	20:		(* Move to idle *)
		uiSignalOutControl := Move_to_idle;
		IF uiSignalInAck = Move_to_idle THEN
			uiSignalOutControl := 0;
			NewState := 25;
		END_IF

	25:
		IF uiSignalInAck = 0 THEN
			NewState := 30;
		END_IF

	30:		(* Set CmdByte to 2, to tell PC to start calibration of Cam 1 *)
		bCalibCamOneStart := TRUE;

		IF stDataFromVision.CmdInProcess =  stDataToVision.CmdByte AND stDataToVision.CmdByte <> 0 THEN							(* When PC recieve command, it sends acknowledge *)
			bCalibCamOneStart := FALSE;
			NewState := 35;
		END_IF
		
	35:
		FB_CLOSE_CUT.Execute := TRUE;
		IF FB_CLOSE_CUT.Done THEN
			FB_CLOSE_CUT.Execute := FALSE;
			NewState := 37;
		END_IF
		
	37:
		IF sNewCalib = 'calib-mounted' THEN
			NewState := 40;
		END_IF
		

	40:		(* Call CALIB_CAM1 on robot Cut. Robot Cut move to a pos to take a picture *)
		uiSignalOutControl := CalibCamOne;
		IF uiSignalInAck = CalibCamOne THEN
			uiSignalOutControl := 0;
			NewState := 45;
		END_IF

	45:
		IF uiSignalInAck = 0 THEN
			NewState := 50;
		END_IF

	50:		(* Before the picture is taken, call get cut coord *)
		getCutCoords := TRUE;										(* Get coord from robot Cut *)
		IF uiSignalInAck = getCurrentCutCoords THEN
			uiSignalOutControl := 0;
			NewState := 55;
		END_IF

	55:
		IF uiSignalInAck = 0 THEN
			bWait := TRUE;
			IF Wait.Q THEN
				bWait := FALSE;
				NewState := 60;
			END_IF
		END_IF

	60:		(* CmdByte 3 means that we want to take a picture *)
		bNewPosCalibCamOne := TRUE;
		IF stDataFromVision.CmdInProcess =  stDataToVision.CmdByte AND stDataToVision.CmdByte <> 0 THEN
			bNewPosCalibCamOne := FALSE;
			NewState := 70;
		END_IF

	70:		(* If there has not been taken enough pictures go to state 40 in order to take more picture. Else send CmdByte 4 to tell PC to stop calib *)
		uiCalibImgCount := uiCalibImgCount + 1;
		IF uiCalibImgCount < 8 THEN
			NewState := 40;
		ELSE
			uiCalibImgCount := 0;
			bEndCalibCamOne := TRUE;
			NewState := 80;
		END_IF

	80:		(* Reset CmdByte and go to init state *)
		uiSignalOutControl := Move_to_idle;
		IF uiSignalInAck = Move_to_idle THEN
			uiSignalOutControl := 0;
			NewState := 82;
		END_IF
	
	82:		
		IF sNewCalib = 'calib-unmounted' THEN
			uiSignalOutTool.06 := FALSE;
			NewState := 84;
		END_IF	
		
	84:
		uiSignalOutControl := Move_to_idle;
		IF uiSignalInAck = Move_to_idle THEN
			uiSignalOutControl := 0;
			NewState := 90;
		END_IF

	85:
		IF uiSignalInAck = 0 THEN
			NewState := 90;
		END_IF

	90:
		IF stDataFromVision.CmdInProcess = stDataToVision.CmdByte AND stDataToVision.CmdByte <>0 THEN
			bEndCalibCamOne := FALSE;
			GbCloseCut := FALSE;
			uiStatus := 0;
			NewState := 0;
		END_IF

	1000:		(* RESET *)
		uiSignalOutTool.06 := FALSE;
		startCalibCam1 			:= FALSE;
		uiSignalOutControl 		:= 0;
		bCalibCamOneStart 		:= FALSE;
		getCutCoords				:= FALSE;
		bNewPosCalibCamOne 	:= FALSE;
		uiCalibImgCount			:= 0;
		bEndCalibCamOne		:= FALSE;

		NewState := 0;

	2000:
		bStopped := TRUE;


END_CASE

IF bStart AND NOT bStop AND NOT bAlarmState AND uiprogNo = 1 AND State <> 2000 THEN
	startCalibCam1 := TRUE;
	(*bStart := FALSE;*)
	uiStatus := 1;
END_IF

IF State <> 2000 THEN
	bStopped := FALSE;
END_IF
Wait		(IN:=  bWait		, PT:=t#1000ms, Q=>, ET=>); 		(*Timer*)
Wait2	(IN:=  bWait2		, PT:=t#2000ms, Q=>, ET=>); 	(*Timer*)
Wait3	(IN:=  bWait3		, PT:=t#2000ms, Q=>, ET=>); 	(*Timer*)

END_PROGRAM

// ---- POUs/CONTROLs/CalibCam2.TcPOU
PROGRAM CalibCam2
VAR_INPUT
	State: INT :=0;
	NewState: INT := 0;
END_VAR

VAR

	Wait: TON;
	Wait2: TON;
	bWait: BOOL;
	bWait2: BOOL;
	next: BOOL;
	Wait3: TON;
	bWait3: BOOL;
	flag: BOOL;
	bStopped: BOOL;
END_VAR

IF sNewCalib = 'he-pick-start' THEN
	startCalibCam2 := TRUE;
ELSE
	startCalibCam2 := FALSE;
END_IF

CASE State OF

	0:		(* Init State - Wait for Calibration of camera 2 *)
		uiSignalOut3.01 := FALSE;
		IF (uiprogNo = 2 OR allZero) AND startCalibCam2 AND State <> 2000  AND NOT bAlarmState THEN
			bWait2 := FALSE;
			uiCalibImgCount := 0;
			uiSignalOut3.01 := TRUE;								(* Tells robot Cut to move to Calib cam 2 pos *)
			startCalibCam2 := FALSE;
			uiSignalOutTool.06 := TRUE;
			flag := FALSE;
			NewState := 10;
		END_IF

	10:		(* Set velocity *)
		uiSignalOutSpeedControl := UINT_TO_BYTE(uiSpeedSetting);
		uiSignalOutControl := Set_Velocity;
		IF uiSignalInAck = Set_Velocity THEN
			uiSignalOutControl := 0;
			NewState := 15;
		END_IF

	15:
		IF uiSignalInAck = 0 THEN
			NewState := 20;
		END_IF

	20:		(* Move to idle *)
		uiSignalOutControl := Move_to_idle;
		IF uiSignalInAck = Move_to_idle THEN
			uiSignalOutControl := 0;
			NewState := 25;
		END_IF

	25:
		IF uiSignalInAck = 0 THEN
			NewState := 27;
		END_IF
		
	27: 		
		FB_CLOSE_CUT.Execute := TRUE;
		IF FB_CLOSE_CUT.Done THEN
			FB_CLOSE_CUT.Execute := FALSE;
			NewState := 29;
		END_IF
	
	29:
		IF sNewCalib = 'calib-mounted' THEN
			NewState := 30;
		END_IF

	30:		(* Move Robot cut to pos for calib *)
		uiSignalOutControl := CalibCamOne;
		IF uiSignalInAck = CalibCamOne THEN
			uiSignalOutControl := 0;
			NewState := 35;
		END_IF

	35:
		IF uiSignalInAck = 0 THEN
			NewState := 40;
		END_IF

	40:		(* Get robot cut pos and orientation *)
		getCutCoords := TRUE;
		IF bPosSentToPcCom AND FB_GET_CUT_COORD.Execute = FALSE THEN
			IF stDataToVision.CoordXR1G <> 0 THEN
				bPosSentToPcCom := FALSE;
				gResetPcCom := TRUE;
				NewState := 45;
			END_IF
		END_IF

	45:
		IF uiSignalInAck = 0 THEN
			GviX	:= stDataToVision.CoordXR1G / 10;
			GviY	:= stDataToVision.CoordYR1G / 10;
			GviZ	:= stDataToVision.CoordZR1G / 10;
			GviA	:= - currentRobotA;
			GviE	:= - currentRobotE;
			GviR	 := 60;
			gResetPcCom := TRUE;

			NewState := 50;
		END_IF

	50:		(* Sends coordinates of calibration board to robot pick *)

		bCalibCamTwoStart := TRUE;
		(* GsendCoord			-->	Starter SendCoordinates sekvensen							-	Sender koordinater til robotterne 		*)
		(* uiSignalOutShared.06	-->	Bekræftelse på at koordinaterne er sendt til udgangene i box 10	-	Acknowledge fra SendCoordinates	*)
		GsendCoord := TRUE;
		IF uiSignalOutShared.06 THEN
			(* Send_pos	-->	Kommando der fortæller robot cut at nogle nye positioner er sendt *)
			uiSignalOutControl := Send_pos;
		END_IF
		IF uiSignalInAck = Send_pos THEN
			uiSignalOutControl := 0;
			NewState := 55;
		END_IF

	55:
		IF uiSignalInAck = 0 THEN
			IF stDataFromVision.CmdInProcess =  stDataToVision.CmdByte AND stDataToVision.CmdByte <> 0 THEN
				bCalibCamTwoStart := FALSE;
				gResetPcCom := TRUE;
				NewState := 60;
			END_IF
		END_IF

	60:		(* Call CALIB_CAM2 on robot Pick. This means that robot Pick move to a pos so that the camera can take a picture *)
		uiSignalOutControl := CalibCamTwo;

		IF uiSignalInAck = CalibCamTwo THEN
			uiSignalOutControl := 0;
			NewState := 65;
		END_IF

	65:
		IF uiSignalInAck = 0 THEN
			NewState := 70;
		END_IF

	70:		(* Before the picture is taken, call get pick coord *)
		getPickCoords := TRUE;
		IF uiSignalInAck = getCurrentPickCoords THEN
			uiSignalOutControl := 0;
			NewState := 75;
		END_IF

	75:
		IF uiSignalInAck = 0 THEN
			bWait2 := TRUE;
			IF Wait2.Q THEN
				bWait2 := FALSE;
				NewState := 80;
			END_IF
		END_IF

	80:		(* CmdByte 6 means that we want to take a picture *)
		IF next5 THEN
			bNewPosCalibCamTwo := TRUE;
			IF stDataFromVision.CmdInProcess =  stDataToVision.CmdByte AND stDataToVision.CmdByte <> 0  THEN
				next5 := FALSE;
				bNewPosCalibCamTwo := FALSE;
				NewState := 85;
			END_IF
		END_IF

	85:		(* If there has not been taken enough pictures go to state 40 in order to take more picture. Else send CmdByte 7 to tell PC to stop calib *)
		uiCalibImgCount := uiCalibImgCount + 1;
		IF uiCalibImgCount < 11 THEN
			gResetPcCom := TRUE;
			NewState := 60;	(* 40 Before *)
		ELSE
			uiCalibImgCount := 0;
			bEndCalibCamTwo := TRUE;
			NewState := 86;
		END_IF
		
	86:
		FB_PICK_TO_IDLE.Execute := TRUE;
		uiSignalOutControl := FB_PICK_TO_IDLE.OutQ;
		IF FB_PICK_TO_IDLE.Done THEN
			FB_PICK_TO_IDLE.Execute := FALSE;
			NewState := 87;
		END_IF
		
	87:
		FB_CUT_TO_IDLE.Execute := TRUE;
		uiSignalOutControl := FB_CUT_TO_IDLE.OutQ;
		IF FB_CUT_TO_IDLE.Done THEN
			IF stDataFromVision.CmdInProcess = stDataToVision.CmdByte  AND stDataToVision.CmdByte <> 0 THEN
				FB_CUT_TO_IDLE.Execute := FALSE;
				bEndCalibCamTwo := FALSE;
				uiStatus := 0;
				uiSignalOutTool.06 := FALSE;
				NewState := 88;
			END_IF
		END_IF
		
	88:
		IF sNewCalib = 'calib-unmounted' THEN
			NewState := 90;
		END_IF	
		

	90:		(* Reset CmdByte and go to init state *)
		//bBackToZero := TRUE;
		uiSignalOutControl := Move_to_idle;
		IF uiSignalInAck = Move_to_idle AND NOT bAck THEN
			uiSignalOutControl := 0;
			IF stDataFromVision.CmdInProcess = stDataToVision.CmdByte  AND stDataToVision.CmdByte <> 0 THEN
				bEndCalibCamTwo := FALSE;
				uiStatus := 0;
				NewState := 95;
			END_IF
		END_IF
		
	95:
		IF uiSignalInAck = 0 THEN
			PcCom.state := 0;
			NewState := 0;
		END_IF

	1000: 		(* RESET *)
		uiSignalOutTool.06 		:= FALSE;
		uiSignalOut3.01 			:= FALSE;
		startCalibCam2 			:= FALSE;
		flag 						:= FALSE;
		uiSignalOutControl 		:= 0;
		getCutCoords 			:= FALSE;
		getPickCoords 			:= FALSE;
		bCalibCamTwoStart 		:= FALSE;
		GcoordSent 				:= FALSE;
		bNewPosCalibCamTwo 	:= FALSE;
		next5 					:= FALSE;
		uiCalibImgCount 			:= 0;
		bEndCalibCamTwo 		:= FALSE;
		bWait2 					:= FALSE;

		NewState := 0;

	2000:
		bStopped := TRUE;


END_CASE

IF bStart AND NOT bStop AND NOT bAlarmState AND uiprogNo = 2 AND State <> 2000 THEN
	startCalibCam2 := TRUE;
	bStart := FALSE;
	uiStatus := 1;
END_IF

IF State <> 2000 THEN
	bStopped := FALSE;
END_IF

Wait		(IN:=  bWait		, PT:=t#200ms, Q=>, ET=>); 		(*Timer*)
Wait2	(IN:=  bWait2		, PT:=t#2000ms, Q=>, ET=>); 	(*Timer*)
Wait3	(IN:=  bWait3		, PT:=t#2000ms, Q=>, ET=>); 	(*Timer*)

END_PROGRAM

// ---- POUs/BackToZero.TcPOU
PROGRAM BackToZero
VAR_INPUT
	State: 		INT := 0;
	NewState:	INT := 0;
END_VAR
VAR
	uiPickCoordX: UINT;
	uiPickCoordY: UINT;
	uiPickCoordZ: UINT;
	
	flag: bool := false;

	StartBackToZero: BOOL;
	bReset: BOOL;
	CANCEL_MOVE: BOOL;
	uiCutCoordX: UINT;
	uiCutCoordY: UINT;
	uiCutCoordZ: UINT;

	timer : TON;
	CoordZR2G: INT;
	PICKMOVED: BOOL;
	CUTMOVED: BOOL;
	whatState: INT;
END_VAR

(* Start connection to Robot Cut if physical botton or HMI button is pressed *)
IF bBackToZero THEN
	StartBackToZero := TRUE;
ELSE
	StartBackToZero := FALSE;
END_IF

CASE State OF

	0:
		IF StartBackToZero THEN
			NewState  	:= 10;
		END_IF

	10:		(* RESET ALL SEQUENCES *)
		IF NOT bReset THEN
			whatState :=  Control.State;
			bReset := TRUE;
			BlockTest.				NewState := 1000;
			Control.					NewState := 1000;
			ControlAuto.				NewState := 1000;
			ControlMoveToCalibPos.	NewState := 1000;
			CalibCam1.				NewState := 1000;
			CalibCam2.				NewState := 1000;
			ControlGrabAuto.			NewState := 1000;

			FB_GET_STEM.			NewState := 1000;
			FB_GRAB_STEM.			NewState := 1000;
			FB_MOVE_ON_STEM.		NewState := 1000;
			FB_FIND_JOINT.			NewState := 1000;
			FB_GRAB_JOINT.			NewState := 1000;
			FB_DELEAF_PLACE.		NewState := 1000;

			getPickCoords 	:= FALSE;
			getCutCoords 	:= FALSE;
		END_IF

		IF Control.NewState = 0 AND ControlAuto.NewState = 0 AND ControlMoveToCalibPos.NewState = 0 AND
			CalibCam1.NewState = 0 AND CalibCam2.NewState = 0 AND ControlGrabAuto.NewState = 0 THEN
			timer.IN := TRUE;
			IF timer.Q THEN
				timer.IN := FALSE;
				bReset := FALSE;
				getPickCoords := FALSE;
				getCutCoords := FALSE;
				NewState := 20;
			END_IF
		END_IF

	20:		(* SEND SIGNAL TO ROBOTS TO STOP MOTION *)
		CANCEL_MOVE := TRUE;
		IF uiSignalInAck = 0 THEN
			timer.IN := TRUE;
			IF timer.Q THEN
				timer.IN := FALSE;
				CANCEL_MOVE := FALSE;
				NewState := 25;
			END_IF
		END_IF
		
	25:		(* Set calibration velocity *)
		uiSignalOutSpeedControl := UINT_TO_BYTE(uiSpeedSetting);
		uiSignalOutControl := Set_Velocity;

		IF uiSignalInAck = Set_Velocity THEN
			uiSignalOutControl := 0;
			NewState := 30;
		END_IF


	30:		(* FIGURE OUT WHICH ROBOT IS SITURATED THE LOWEST *)
		(* Get Cut coord *)
		getCutCoords := TRUE;
		IF bPosSentToPcCom AND FB_GET_CUT_COORD.Execute = FALSE THEN
			bPosSentToPcCom := FALSE;
			gResetPcCom := TRUE;
			NewState := 35;
		END_IF

	35:
		IF uiSignalInAck = 0 THEN
			uiCutCoordX	:= stDataToVision.CoordXR1G / 10;
			uiCutCoordY	:= stDataToVision.CoordYR1G / 10;
			uiCutCoordZ	:= stDataToVision.CoordZR1G / 10;
			timer.IN := TRUE;
			IF timer.Q THEN
				timer.IN := FALSE;
				gResetPcCom := TRUE;
				NewState := 40;
			END_IF
		END_IF


	40:
		(* Get Cut coord *)
		getPickCoords := TRUE;
		IF bPosSentToPcCom AND FB_GET_PICK_COORD.Execute = FALSE THEN
			bPosSentToPcCom := FALSE;
			gResetPcCom := TRUE;
			NewState := 45;
		END_IF

	45:
		IF uiSignalInAck = 0 THEN
			uiPickCoordX	:= stDataToVision.CoordXR2G / 10;
			uiPickCoordY	:= stDataToVision.CoordYR2G / 10;
			uiPickCoordZ	:= stDataToVision.CoordZR2G / 10;
			timer.IN := TRUE;
			IF timer.Q THEN
				timer.IN := FALSE;
				gResetPcCom := TRUE;
				NewState := 50;
			END_IF
		END_IF
		
	50:		(* MOVE THE FIRST ROBOT AWAY *)
		IF whatState >= 400 AND whatState <=500 THEN
			FB_PICK_TO_ZERO.Execute := TRUE;
			uiSignalOutControl := FB_PICK_TO_ZERO.OutQ;
			IF FB_PICK_TO_ZERO.Done THEN
				PICKMOVED := TRUE;
				FB_PICK_TO_ZERO.Execute := FALSE;
				NewState := 60;
			END_IF
		ELSE
			FB_CUT_TO_ZERO.Execute := TRUE;
			uiSignalOutControl := FB_CUT_TO_ZERO.OutQ;
			IF FB_CUT_TO_ZERO.Done THEN
				CUTMOVED := TRUE;
				FB_CUT_TO_ZERO.Execute := FALSE;
				NewState := 60;
			END_IF
		END_IF

	60:		(* MOVE THE LAST ROBOT *)
		IF PICKMOVED THEN
			FB_CUT_TO_ZERO.Execute := TRUE;
			uiSignalOutControl := FB_CUT_TO_ZERO.OutQ;
			IF FB_CUT_TO_ZERO.Done THEN
				FB_CUT_TO_ZERO.Execute := FALSE;
				NewState := 70;
			END_IF
		ELSE
			FB_PICK_TO_ZERO.Execute := TRUE;
			uiSignalOutControl := FB_PICK_TO_ZERO.OutQ;
			IF FB_PICK_TO_ZERO.Done THEN
				FB_PICK_TO_ZERO.Execute := FALSE;
				NewState := 70;
			END_IF
		END_IF

	(*50:		(* MOVE THE LOWEST ROBOT AWAY *)
		IF uiCutCoordZ < (uiPickCoordZ - 20) THEN
			FB_CUT_TO_ZERO.Execute := TRUE;
			uiSignalOutControl := FB_CUT_TO_ZERO.OutQ;
			IF FB_CUT_TO_ZERO.Done THEN
				FB_CUT_TO_ZERO.Execute := FALSE;
				NewState := 60;
			END_IF
		ELSE
			FB_PICK_TO_ZERO.Execute := TRUE;
			uiSignalOutControl := FB_PICK_TO_ZERO.OutQ;
			IF FB_PICK_TO_ZERO.Done THEN
				FB_PICK_TO_ZERO.Execute := FALSE;
				NewState := 60;
			END_IF
		END_IF

	60:		(* MOVE THE LAST ROBOT *)
		IF uiCutCoordZ > (uiPickCoordZ - 20) THEN
			FB_CUT_TO_ZERO.Execute := TRUE;
			uiSignalOutControl := FB_CUT_TO_ZERO.OutQ;
			IF FB_CUT_TO_ZERO.Done THEN
				FB_CUT_TO_ZERO.Execute := FALSE;
				NewState := 70;
			END_IF
		ELSE
			FB_PICK_TO_ZERO.Execute := TRUE;
			uiSignalOutControl := FB_PICK_TO_ZERO.OutQ;
			IF FB_PICK_TO_ZERO.Done THEN
				FB_PICK_TO_ZERO.Execute := FALSE;
				NewState := 70;
			END_IF
		END_IF*)

	70:		(* MOVE BACK TO IDLE *)
		FB_MOVE_TO_IDLE.Execute := TRUE;
		uiSignalOutControl := FB_MOVE_TO_IDLE.OutQ;
		IF FB_MOVE_TO_IDLE.Done THEN
			FB_MOVE_TO_IDLE.Execute := FALSE;
			NewState := 80;
		END_IF


	80:		(* RESET THE TOOLS *)
		IF flag = FALSE THEN
			Tools.NewState := 1000;
			flag := TRUE;
		END_IF
		
		IF uiToolState = 0 THEN
			flag := false;
			NewState := 90;
		END_IF


	90:		(* RESET VALUES AND CHANGE STATE TO 0 *)
		bBackToZero := FALSE;
		CANCEL_MOVE := FALSE;
		PICKMOVED := FALSE;
		CUTMOVED := FALSE;
		whatState := 0;

		uiCutCoordX	:= 0;
		uiCutCoordY	:= 0;
		uiCutCoordZ 	:= 0;
		uiPickCoordX	:= 0;
		uiPickCoordY := 0;
		uiPickCoordZ := 0;
		gStopped := TRUE;
		NewState := 0;


END_CASE

uiSignalOut2.03 := CANCEL_MOVE;
 timer( PT:=t#500ms, Q=>, ET=>);

END_PROGRAM

// ---- POUs/CONTROLs/BlockTest.TcPOU
PROGRAM BlockTest
VAR_INPUT
	State: INT := 0;
	NewState: INT := 0;

	InternalState: INT := 0;
	InternalNewState: INT := 0;
END_VAR

VAR
	(* FUNCTION BLOCKS *)
	(*FB_PLACE: 		PlaceCoordinates;
	FB_GET_STEM:	GetStem;*)

	(* REALS *)

	(* INTEGERS *)


	ImageRetryHeight:	INT;

	iMoved: 			INT;					(* Hvor mange gange har cut bevæget sig efter iBunchPosZ er nået *)
	iCnfgChange:		INT := 0;
	uiDeleaf: 		UINT;

	(* BOOLS *)
	bStopped: BOOL;
	bRobotFail: BOOL;

	bRetry: INT;
	bStemGrabbed: BOOL;

END_VAR

CASE State OF

	0:		(* init	-	Every important variables will be resat before the start of the sequence *)
		IF bStart AND uiprogNo = 7 AND State <> 2000  AND NOT bAlarmState THEN
			uiStatus := 1;

			(* Init variables *)
			bRetry := 0;
			uiCalibImgCount	:= 0;
			iMoved := 0;
			iImageZone := 0;
			gJointFound := 0;
			gResetPcCom 	:= TRUE;
			iCnfgChange := 0;
			uiDeleaf := 0;
			bPosSentToPcCom := FALSE;

			(* Before starting - Home *)
			GbHomeGripStem := TRUE;
			IF bHomeDone THEN
				bStart := FALSE;
				bHomeDone := FALSE;
				NewState := 10;
			END_IF
		END_IF

	10:		(* Set velocity *)
		FB_SET_VELOCITY.Execute := TRUE;
		uiSignalOutSpeedControl := UINT_TO_BYTE(uiSpeedSetting);
		uiSignalOutControl := FB_SET_VELOCITY.OutQ;
		IF FB_SET_VELOCITY.Done THEN
			FB_SET_VELOCITY.Execute := FALSE;
			NewState := 20;
		END_IF

	20:		(* Idle *)
		FB_MOVE_TO_IDLE.Execute := TRUE;
		uiSignalOutControl := FB_MOVE_TO_IDLE.OutQ;
		IF FB_MOVE_TO_IDLE.Done THEN
			FB_MOVE_TO_IDLE.Execute := FALSE;
			NewState := 30;
		END_IF




		(* ------------------------------------------------------------------- Get Stem  ------------------------------------------------------------------- *)
	30:				(*  Load cutter *)
		FB_LOAD_CUT.Execute := TRUE;
		IF FB_LOAD_CUT.Done THEN
			FB_LOAD_CUT.Execute := FALSE;
			NewState := 40;
		END_IF


		(* Get stem SEQUENCE *)
	40:
		FB_GET_STEM.Execute := TRUE;
		IF FB_GET_STEM.Done THEN
			IF FB_GET_STEM.Fail THEN
				FB_GET_STEM.Execute := FALSE;
				bBackToZero := TRUE;
			ELSE
				FB_GET_STEM.Execute := FALSE;
				NewState := 100;
			END_IF
		END_IF











	(* ------------------------------------------------------------------- Grab Stem  ------------------------------------------------------------------- *)
	100:
		FB_GRAB_STEM.Execute := TRUE;
		IF FB_GRAB_STEM.Done THEN
			IF FB_GRAB_STEM.Fail THEN
				FB_GRAB_STEM.Execute := FALSE;
				bBackToZero := TRUE;
			ELSE
				FB_GRAB_STEM.Execute := FALSE;
				NewState := 200;
			END_IF
		END_IF










	(* ------------------------------------------------------------------- Move On Stem  ------------------------------------------------------------------- *)
	200:
		FB_MOVE_ON_STEM.Execute := TRUE;
		IF FB_MOVE_ON_STEM.Done THEN
			IF FB_MOVE_ON_STEM.Fail THEN
				bBackToZero := TRUE;
				FB_MOVE_ON_STEM.Execute := FALSE;
			ELSIF FB_MOVE_ON_STEM.JointReached THEN
				FB_MOVE_ON_STEM.Execute := FALSE;
				(* Grabbing sequence *)
				gResetPcCom := TRUE;
				IF uimodeNo <= 1 THEN
					NewState := 400;
				ELSE
					NewState := 420;
				END_IF
			ELSE
				FB_MOVE_ON_STEM.Execute := FALSE;
				NewState := 300;
			END_IF
		END_IF












	(* ------------------------------------------------------------------- Find Joint  ------------------------------------------------------------------- *)
	300:
		FB_FIND_JOINT.Execute := TRUE;
		IF FB_FIND_JOINT.Done THEN
			IF FB_FIND_JOINT.Fail THEN
				FB_FIND_JOINT.Execute := FALSE;
				bBackToZero := TRUE;
			ELSE
				FB_FIND_JOINT.Execute := FALSE;
				NewState := 400;
			END_IF
		END_IF



	(* ------------------------------------------ Grab tomatoes ------------------------------------------ *)
	400:		(* Robot Pick grab *)

		FB_GRAB_JOINT.Execute := TRUE;
		IF FB_GRAB_JOINT.Done THEN
			IF FB_GRAB_JOINT.bRetry <> 0 THEN
				FB_GRAB_JOINT.Execute := FALSE;
				NewState := 300;
			ELSIF FB_GRAB_JOINT.Fail THEN
				FB_GRAB_JOINT.Execute := FALSE;
				bBackToZero := TRUE;
			ELSE
				FB_GRAB_JOINT.Execute := FALSE;
				NewState := 500;
			END_IF
		END_IF



	(* --------------------------------- DELEAFING ------------------------------------ *)
	500:
		FB_DELEAF_PLACE.Execute := TRUE;
		IF FB_DELEAF_PLACE.Done THEN
			FB_DELEAF_PLACE.Execute := FALSE;
			NewState := 600;
		END_IF


	600:		(*Open Cut*)
		FB_OPEN_CUT.Execute := TRUE;
		IF FB_OPEN_CUT.Done THEN
			FB_OPEN_CUT.Execute := FALSE;
			NewState := 610;
		END_IF

	610:		(*Move cut away from stem*)
		FB_CUT_FROM_STEM.Execute := TRUE;
		uiSignalOutControl := FB_CUT_FROM_STEM.OutQ;
		IF FB_CUT_FROM_STEM.Done THEN
			FB_CUT_FROM_STEM.Execute := FALSE;
			NewState := 620;
		END_IF


	620:		(* GbReleaseStem *)
		(* Grab stem and pull in *)
		IF NOT bAck THEN
			(* HMI knap der kalder GribStem *)
			GbReleaseStem := TRUE;
		ELSIF bAck THEN
			NewState := 630;
		END_IF

	630:		(* Move to idle *)
		FB_MOVE_TO_IDLE.Execute := TRUE;
		uiSignalOutControl := FB_MOVE_TO_IDLE.OutQ;
		IF FB_MOVE_TO_IDLE.Done THEN
			FB_MOVE_TO_IDLE.Execute := FALSE;
			uiStatus := 0;
			NewState := 640;
		END_IF

	640:		(* Deload *)

		FB_DELOAD_CUT.Execute := TRUE;
		IF FB_DELOAD_CUT.Done THEN
			FB_DELOAD_CUT.Execute := FALSE;
			NewState := 0;
		END_IF




	1000:	(* Reset *)

		uiSignalOutControl  := 0;		(* Stop sequences on ROBOTS *)

		(* Reset timers *)
		bRetry := 0;
		stDataToVision.ResultRead := 1;
		gResetPcCom := TRUE;
		iCnfgChange := 1;
		uiCalibImgCount := 0;
		uiDeleaf := 0;
		InternalNewState := 0;
		NewState := 0;

	2000:
		bStopped := TRUE;


	(* ----------------------------- FAILED WHEN MOVING ON STEM ----------------------------- *)
	3000:		(* First figure out if cut is under the lowest tomato *)
		(* Get Cut coord *)
		getCutCoords := TRUE;
		IF bPosSentToPcCom AND FB_GET_CUT_COORD.Execute = FALSE THEN
			bPosSentToPcCom := FALSE;
			gResetPcCom := TRUE;
			NewState := 3005;
		END_IF

	3005:
		IF uiSignalInAck = 0 THEN
			uiCutCoordX	:= stDataToVision.CoordXR1G / 10;
			uiCutCoordY	:= stDataToVision.CoordYR1G / 10;
			uiCutCoordZ	:= stDataToVision.CoordZR1G / 10;

			NewState := 3010;
		END_IF

	3010:

		IF uiCutCoordZ > iBunchPosZ THEN
			(* Then cut must have reached the joint*)
			NewState := 330;

		ELSE
			(* It must be a too big of a stick-out *)
			FB_RELEASE_CUT.Execute := TRUE;
			IF FB_RELEASE_CUT.Done THEN
				FB_RELEASE_CUT.Execute := FALSE;
				NewState := 3020;
			END_IF
		END_IF

	3020:
		FB_LOAD_CUT.Execute := TRUE;
		IF FB_LOAD_CUT.Done THEN
			FB_LOAD_CUT.Execute := FALSE;
			NewState := 320;
		END_IF



END_CASE

IF State <> 2000 THEN
	bStopped := FALSE;
END_IF

bRobotFail := uiSignalIn2.07;

END_PROGRAM

// ---- POUs/RobotService.TcPOU
PROGRAM RobotService
VAR_INPUT
	State: 		INT := 0;
	NewState:	INT := 0;
END_VAR
VAR


	timer : TON;
END_VAR



CASE State OF

	0:
		IF bRobotServiceStart THEN
			NewState  	:= 10;
		END_IF

	10:		(* Reset the tools *)
		Tools.NewState := 1000;
		IF Tools.NewState = 0 THEN
			NewState := 20;
		END_IF

	20:
		FB_ROBOT_SERVICE.Execute := TRUE;
		uiSignalOutControl := FB_ROBOT_SERVICE.Command;
		IF FB_ROBOT_SERVICE.Done THEN
			FB_ROBOT_SERVICE.Execute := FALSE;
			NewState := 30;
		END_IF

	30:
		IF bRobotServiceStop THEN
			NewState := 40;
		END_IF

	40:
		FB_MOVE_TO_IDLE.Execute := TRUE;
		uiSignalOutControl := FB_MOVE_TO_IDLE.Command;
		IF FB_MOVE_TO_IDLE.Done THEN
			FB_MOVE_TO_IDLE.Execute := FALSE;
			uiSignalOutControl := 0;
			NewState := 0;
		END_IF


	90:		(* RESET VALUES AND CHANGE STATE TO 0 *)



		NewState := 0;


END_CASE

END_PROGRAM

// ---- POUs/FUNCTIONs/RobotControl_1.TcPOU
FUNCTION_BLOCK RobotControl_1
VAR_INPUT
	ControlType: 	USINT;		(*	1: Controlling valves from Robot		2: Controlling valves from Robot and  PLC		3: Close only using PLC		4: Open only using PLC		*)
	Command:	USINT;		(*	Command to Robot		*)
	Ack: 		BYTE;		(*	Acknowledge from Robot	*)
	Execute: 		BOOL;

	CoordX:		INT;
	CoordY:		INT;
	CoordZ:		INT;

END_VAR
VAR_OUTPUT
	OutQ: 		BYTE;
END_VAR
VAR
	trigger : 		R_TRIG;
	R_Execute : 	R_TRIG;
	WaitValve:	TON;

	State : INT;
	NewState : INT;

	Done: 		BOOL;
	bValveTime: 	BOOL;
END_VAR

IF State <> NewState THEN
	State := NewState;
END_IF

CASE  State OF
	0:
		Done := FALSE;
		IF Execute  THEN
			IF ControlType = 1 THEN
				NewState	 :=10;
			ELSIF ControlType = 2 THEN
				NewState := 50;
			ELSE
				NewState := 0;
			END_IF
		END_IF

	10:
		(* Send command To robot *)
		OutQ := Command;
		(* When Robot sends back the same command, the command starts *)
		IF Ack = Command THEN
			OutQ := 0;
			NewState := 20;
		END_IF

	20:
		(* When Ack is 0, the command has been executed *)
		IF Ack = 0 THEN
			NewState := 1000;
		END_IF

	50:
		IF CoordX = 0 AND CoordY = 0 AND CoordZ = 0 OR OutQ = Command THEN
			OutQ := Command;
			IF Ack = Command THEN
				OutQ := 0;
				NewState := 20;
			END_IF
		END_IF


	1000:
		Done := TRUE;
		IF NOT Execute THEN
			NewState := 0;
		END_IF



END_CASE

END_FUNCTION_BLOCK

// ---- POUs/FUNCTIONs/CamControl_1.TcPOU
FUNCTION_BLOCK CamControl_1
VAR_INPUT
	NewState : 	INT;
	ControlType: 	USINT;		(*	1: Controlling valves from Robot		2: Controlling valves from Robot and  PLC		3: Close only using PLC		4: Open only using PLC		*)
	CommandNo:	USINT;		(*	Command to Robot		*)
	Ack: 		BYTE;		(*	Acknowledge from Robot	*)
	Execute: 		BOOL;

	TrunkPosX:		INT;
	TrunkPosY:		INT;			(*	Distance to the stem 					*)
	TrunkPosZ:		INT;
	BunchPosX:		INT;
	BunchPosY:		INT;
	BunchPosZ:		INT;			(*	The height of the lowest hangiung tomato	*)
	StemAngle:		INT;
END_VAR
VAR_OUTPUT
	TrunkDist:		INT;			(*	Distance to the stem 					*)
	BunchHeight:		INT;			(*	The height of the lowest hangiung tomato	*)
	StemHeading:	INT;
	X:				INT;
	Y:				INT;
	Z: 				INT;

	Zone:			USINT;

	Command:		BOOL;
END_VAR
VAR
	trigger : 		R_TRIG;
	R_Execute : 	R_TRIG;
	Wait:		TON;

	State : 		INT;
	
	Offset:		INT := 220;

	Done: 		BOOL;
	bValveTime: 	BOOL;
	Retry: BOOL;
	Fail: BOOL;
END_VAR

IF State <> NewState THEN
	State := NewState;
END_IF

CASE  State OF
	0:
		Done := FALSE;
		IF Execute  THEN
			IF ControlType = 1 THEN
				NewState	 :=10;
			ELSIF ControlType = 2 THEN
				NewState := 50;
			ELSE
				NewState := 0;
			END_IF
		END_IF

	10:		(* Send CmdByte  to PC	-	Stationary cam takes picture *)
		Wait.IN := FALSE;
		Command := TRUE;
		IF CommandNo = Ack AND Ack <> 0 THEN			(* When the PC  has sent the position, prepare to send the position to robot pick *)
			IF (TrunkPosY > 600  OR BunchPosY > 600 OR TrunkPosY < 100 OR BunchPosY < 100 OR TrunkPosX > 500) AND NOT Retry THEN
				Command := FALSE;
				NewState := 30;
			ELSIF (TrunkPosY > 600  OR BunchPosY > 600 OR TrunkPosY < 100 OR BunchPosY < 100 OR TrunkPosX > 500) AND Retry THEN
				Command := FALSE;
				Fail := TRUE;
				NewState := 1000;
			ELSE
				Retry := FALSE;
				(* uiTrunkPos		-->	Distance to trunk in mm								 	-								*)
				(* uiDistToGrab	-->	Tells Tools program how far Grip has to move				-	Global Variabel Tool looks at	*)
				(* uiGripOffset		-->	Distance from Workframe Y=0 to grip Y pos 												*)
				TrunkDist := TrunkPosY - Offset;

				(* iBunchPosZ	-->	The height will be used to know how far to move before looking for joint							*)
				BunchHeight := BunchPosZ;
				StemHeading := StemAngle;

				X := BunchPosX;
				Y := BunchPosY;
				Z := BunchPosZ;
	
				IF (StemHeading < -125 AND StemHeading >=-180) OR (StemHeading >135 AND StemHeading < 180) THEN
					Zone := 1;
				ELSIF (StemHeading <= 135 AND StemHeading >= 35) THEN
					Zone := 2;
				ELSIF (StemHeading >= -125 AND StemHeading <= -45) THEN
					Zone := 3;
				ELSIF (StemHeading > -45 AND StemHeading < 35) THEN
					Zone := 4;
				ELSE
					Zone := 0;
				END_IF
	
				Command := FALSE;
				NewState := 20;

			END_IF
		END_IF

	20:
		(* When Ack is 0, the command has been executed *)
		IF Ack = 0 THEN
			NewState := 1000;
		END_IF
	30:
		IF Wait.Q THEN
			Retry := TRUE;
			NewState := 10;
		END_IF

	1000:
		Done := TRUE;
		IF NOT Execute THEN
			Fail := FALSE;
			Retry := FALSE;
			NewState := 0;
		END_IF



END_CASE

Wait		(IN:=  State = 30		, PT:=t#500ms, Q=>, ET=>); 		(*Timer*)		(* For waiting for Valves 			*)

END_FUNCTION_BLOCK

// ---- POUs/FUNCTIONs/CamControl_2.TcPOU
FUNCTION_BLOCK CamControl_2
VAR_INPUT
		NewState : 	INT;
	X:				INT;
	Y:				INT;
	Z:				INT;
	RotZ0:			INT;
	RotY:			UINT;
	RotZ1:			INT;
	StemHeading:	INT;

	StemFound:		USINT;
	JointFound:		USINT;
	TomatoFound:   	USINT;
	TrussFound:		USINT;

	ControlType: 		USINT;		(*	1: Controlling valves from Robot		2: Controlling valves from Robot and  PLC		3: Close only using PLC		4: Open only using PLC		*)
	CommandNo:		USINT;		(*	Command to Robot		*)
	Ack: 			BYTE;		(*	Acknowledge from Robot	*)
	Execute: 			BOOL;
END_VAR
VAR_OUTPUT
	Command:		BOOL;
	Zone:			USINT;
	PickAngle:		INT;
END_VAR
VAR
	State : 		INT;


	Done: 		BOOL;
	Fail:			BOOL;
	Retry: BOOL;
END_VAR

IF State <> NewState THEN
	State := NewState;
END_IF

CASE  State OF
	0:
		Done := FALSE;
		IF Execute  THEN
			IF ControlType = 1 THEN
				NewState	 :=10;
			ELSIF ControlType = 2 THEN
				NewState := 50;
			ELSE
				NewState := 0;
			END_IF
		END_IF

	10:		(* Send CmdByte  to PC	-	Stationary cam takes picture *)
		Command := TRUE;							(* Send CmdByte 14 to PC *)
		IF CommandNo = Ack AND Ack <> 0 THEN		(* When the PC  has sent the position, prepare to send the position to robot pick *)
			(* Check if the positions are acceptable *)
			IF (X < 100 OR X > 450 OR Y < 100 OR Y > 450 OR Z < 250) AND NOT Retry THEN
				Command := FALSE;
				NewState := 30;
			(* If positions are not acceptable second time, return FAIL := TRUE *)
			ELSIF (X < 100 OR X > 450 OR Y < 100 OR Y > 450 OR Z < 250) AND Retry THEN
				Command := FALSE;
				Retry := FALSE;
				Fail := TRUE;
				NewState := 1000;
			ELSE
				(* Define Zone *)
				IF StemHeading <> 0 THEN
					IF (StemHeading < -125 AND StemHeading >=-180) OR (StemHeading >135 AND StemHeading <= 180) THEN
						Zone := 1;
						IF StemHeading < 0 THEN
							PickAngle := REAL_TO_INT(190 + StemHeading);
							IF StemHeading >= -140 THEN
								PickAngle := REAL_TO_INT(-(190 + StemHeading));		(* IKKE RIGTIGT*)
							END_IF
						ELSE
							PickAngle := REAL_TO_INT(StemHeading - 190);
						END_IF
					ELSIF (StemHeading <= 135 AND StemHeading >= 35) THEN
						Zone := 2;
						PickAngle := REAL_TO_INT(( - 170 + StemHeading ));
					ELSIF (StemHeading >= -125 AND StemHeading <= -45) THEN
						Zone := 3;
						PickAngle := REAL_TO_INT((StemHeading));
					ELSIF (StemHeading > -45 AND StemHeading < 40) THEN
						Zone := 4;
						PickAngle := REAL_TO_INT(StemHeading - 1);
						IF StemHeading < 0 THEN
							PickAngle := REAL_TO_INT(-StemHeading + 1);
						END_IF
					ELSE
						Zone := 0;
					END_IF
				END_IF
				Command := FALSE;
				NewState := 20;
			END_IF
		END_IF

	20:
		(* When Ack is 0, the command has been executed *)
		IF Ack = 0 THEN
			NewState := 1000;
		END_IF

	30:
		Retry := TRUE;
		NewState := 10;

	1000:
		Done := TRUE;
		IF NOT Execute THEN
			Retry := FALSE;
			Fail := FALSE;
			NewState := 0;
		END_IF



END_CASE

END_FUNCTION_BLOCK

// ---- POUs/SEQUENCEs/GetStem.TcPOU
FUNCTION_BLOCK GetStem
VAR_INPUT
	Execute: 		BOOL;
	State : 		INT;
	NewState : 	INT;

END_VAR
VAR_OUTPUT


END_VAR
VAR

	Done: 		BOOL;
	Fail: BOOL;
	bRetry: BOOL;
END_VAR

IF State <> NewState THEN
	State := NewState;
END_IF

CASE  State OF
	0:
		Done := FALSE;
		IF Execute  THEN
			NewState	 :=10;
		END_IF

	10:		(* Cam 1 Take image	-	parameters recieved from Vision = height of lowest ripe tomato and Y coord for lowest point of the stem *)

		FB_CAM_ONE_CONTROL.Execute := TRUE;
		IF FB_CAM_ONE_CONTROL.Done THEN
			FB_CAM_ONE_CONTROL.Execute := FALSE;
			IF FB_CAM_ONE_CONTROL.Fail THEN
				(* Adjust cart height  in order to retry *)
				Fail := TRUE;
				NewState := 1000;
			ELSE
				(* uiDistToGrab 	-->		Distance from Joris Gripper to stem 			*)
				uiDistToGrab	:= FB_CAM_ONE_CONTROL.TrunkDist;
				(* iBunchPosZ	-->		Height of the lowest hanging red tomato		*)
				iBunchPosZ 	:= FB_CAM_ONE_CONTROL.BunchHeight;
				(* i StemAngle	-->		Heading direction from stem to lowest tomato	*)
				iStemAngle	:= FB_CAM_ONE_CONTROL.StemHeading;
				(* iImageZone	-->		Zone of lowest tomato						*)
				iImageZone	:= FB_CAM_ONE_CONTROL.Zone;
				NewState := 20;
			END_IF
		END_IF


	20:				(* Joris gripper retreives stem *)
		(* Grab stem and pull in *)
		IF NOT bAck THEN
			(* HMI knap der kalder GribStem *)
			GbGripStem := TRUE;
		ELSIF bAck THEN
			gResetPcCom := TRUE;
			NewState := 25;
		END_IF

	25:
		(* Needs an option To move cart a bit, to take a new photo *)
		IF uiToolState = 0 THEN
			IF bJorisSensor AND bRetry < 1 THEN
				uiDistToGrab := uiDistToGrab + 50;
				bRetry := 1;
				NewState := 30;
			ELSIF bJorisSensor AND bRetry >= 1 THEN
				Fail := TRUE;
				gResetPcCom := TRUE;
				NewState := 1000;
			ELSE
				bRetry := 0;
				gResetPcCom := TRUE;
				NewState := 1000;
			END_IF
		END_IF

	30:	(* Open gripper *)
		FB_OPEN_GRIP.Execute := TRUE;
		IF FB_OPEN_GRIP.Done THEN
			FB_OPEN_GRIP.Execute := FALSE;
			NewState := 20;
		END_IF


	1000:
		Done := TRUE;
		IF NOT Execute THEN
			Fail := FALSE;
			NewState := 0;
		END_IF



END_CASE

END_FUNCTION_BLOCK

// ---- POUs/SEQUENCEs/GrabStem.TcPOU
FUNCTION_BLOCK GrabStem
VAR_INPUT
	Execute: 		BOOL;
	State : 		INT;
	NewState : 	INT;

END_VAR
VAR_OUTPUT


END_VAR
VAR


	Done: 		BOOL;
	Fail: BOOL;
	bRetry: USINT;
	bRobotFail: BOOL;
END_VAR

IF State <> NewState THEN
	State := NewState;
END_IF

CASE  State OF
	0:
		Done := FALSE;
		IF Execute  THEN
			NewState	 :=10;
		END_IF

	10:		(* Robot Pick move to Image Pos *)
		FB_PICK_TRUNK_IMAGE.Execute := TRUE;
		uiSignalOutControl := FB_PICK_TRUNK_IMAGE.OutQ;
		IF FB_PICK_TRUNK_IMAGE.Done THEN
			FB_PICK_TRUNK_IMAGE.Execute := FALSE;
			gResetPcCom := TRUE;
			NewState := 20;
		END_IF

	20:		(* Send Robot Pick Position *)
		getPickCoords := TRUE;
		IF bPosSentToPcCom AND FB_GET_PICK_COORD.Execute = FALSE THEN
			ImageRetryHeight := stDataToVision.CoordZR2G;
			bPosSentToPcCom := FALSE;
			bGetCoordDone := FALSE;
			NewState := 40;
		END_IF

	40:		(* Cam 2 take image *)
		(* Take bottom Image *)
		(* If pick coordinates are recieved, take an image *)
		IF stDataToVision.CoordXR2G <> 0 AND stDataToVision.CoordYR2G <> 0 AND stDataToVision.CoordZR2G <> 0 THEN
			FB_CAM_TWO_CONTROL.Execute := TRUE;
			IF FB_CAM_TWO_CONTROL.Done THEN
				(* If the positions was unacceptable  - Prepare to take a new picture from 50 mm further up *)
				IF FB_CAM_TWO_CONTROL.Fail THEN
					(* Send new pos to Robots *)
					GviX	:= stDataToVision.CoordXR2G / 10;
					GviY 	:= stDataToVision.CoordYR2G / 10;
					GviZ 	:= (stDataToVision.CoordZR2G / 10) + 50;

					(* GsendCoord			-->	Starter SendCoordinates sekvensen							-	Sender koordinater til robotterne 		*)
					(* uiSignalOutShared.06	-->	Bekræftelse på at koordinaterne er sendt til udgangene i box 10	-	Acknowledge fra SendCoordinates	*)
					GsendCoord := TRUE;
					IF uiSignalOutShared.06 THEN
						(* Send_pos	-->	Kommando der fortæller robot cut at nogle nye positioner er sendt *)
						uiSignalOutControl := Send_pos;
					END_IF
					IF uiSignalInAck = Send_pos THEN
						FB_CAM_TWO_CONTROL.Execute := FALSE;
						uiSignalOutControl := 0;
						uiCalibImgCount := uiCalibImgCount + 1;
						NewState := 50;
					END_IF
				ELSE
					(* If positions are acceptable and stem is found, Send the posiotions to the robots *)
					FB_CAM_TWO_CONTROL.Execute := FALSE;
					IF stDataFromVision.gStemFound = 1 THEN
						GviX	:= FB_CAM_TWO_CONTROL.X;
						GviY 	:= FB_CAM_TWO_CONTROL.Y;
						GviZ 	:= FB_CAM_TWO_CONTROL.Z;
						GviA 	:= FB_CAM_TWO_CONTROL.RotZ0;
						GviE 	:= FB_CAM_TWO_CONTROL.RotY;
						GviR 	:= FB_CAM_TWO_CONTROL.RotZ1;

						GviX2 	:= FB_CAM_TWO_CONTROL.X;
						GviY2 	:= (FB_CAM_TWO_CONTROL.Y + FB_CAM_TWO_CONTROL.Y + FB_CAM_ONE_CONTROL.Y)/3;
						GviZ2 	:= FB_CAM_ONE_CONTROL.Z + 50;

						iImageZone	:= FB_CAM_ONE_CONTROL.Zone;
						NewState := 60;
					(* IF the stem cannot be found, retry grabbing the stem with Joris gripper *)
					ELSE
						IF bRetry = 0 THEN
							bRetry := 1;
							gResetPcCom := TRUE;
							NewState := 20;
						ELSE
							Fail := TRUE;
							NewState := 1000;
						END_IF
					END_IF
				END_IF
			END_IF
		(*ELSE
			gResetPcCom := TRUE;
			NewState := 20;*)
		END_IF


	50:
		IF uiSignalInAck = 0 THEN
			IF bRetry = 0 THEN
				bRetry := bRetry + 1;
				NewState := 10;
			ELSE
				Fail := TRUE;
				NewState := 1000;
			END_IF
		END_IF

	60:		(* Send Pos to Robot *)

		(* GsendCoord			-->	Starter SendCoordinates sekvensen							-	Sender koordinater til robotterne 		*)
		(* uiSignalOutShared.06	-->	Bekræftelse på at koordinaterne er sendt til udgangene i box 10	-	Acknowledge fra SendCoordinates	*)
		GsendCoord := TRUE;
		IF uiSignalOutShared.06 THEN
			(* Send_pos	-->	Kommando der fortæller robot cut at nogle nye positioner er sendt *)
			uiSignalOutControl := Send_two_pos;
		END_IF

		IF uiSignalInAck = Send_two_pos THEN
			uiSignalOutControl := 0;
			uiCalibImgCount := uiCalibImgCount + 1;
			NewState := 65;
		END_IF

	65:
		IF uiSignalInAck = 0 THEN
			NewState := 70;
		END_IF

	70:		(* Grab the stem + Move to image pos *)
		FB_IMAGE_GRAB.Execute := TRUE;
		uiSignalOutControl := FB_IMAGE_GRAB.OutQ;

		IF FB_IMAGE_GRAB.Done THEN
			FB_IMAGE_GRAB.Execute := FALSE;
			NewState := 80;
		END_IF

	80:
		IF NOT bRobotFail THEN
			bRetry := 0;
			gResetPcCom := TRUE;
			NewState := 1000;
		ELSE
			(* Retries:																						*)
			(* Open and close cone								-	To check if it was a misreading from sensor 	*)
			(* Move to pos 50mm above normal image pos, then retry												*)
			IF bRetry  < 2 THEN
				bRetry := bRetry + 1;
				(*uiCalibImgCount := 0;*)
				GviZ2 := stDataToVision.CoordZR2G/10 + 100;
				NewState := 90;
			ELSE
				bBackToZero := TRUE;
			END_IF
		END_IF


	90:
		(* GsendCoord			-->	Starter SendCoordinates sekvensen							-	Sender koordinater til robotterne 		*)
		(* uiSignalOutShared.06	-->	Bekræftelse på at koordinaterne er sendt til udgangene i box 10	-	Acknowledge fra SendCoordinates	*)
		GsendCoord := TRUE;
		IF uiSignalOutShared.06 THEN
			(* Send_pos	-->	Kommando der fortæller robot cut at nogle nye positioner er sendt *)
			uiSignalOutControl := Send_two_pos;
		END_IF

		IF uiSignalInAck = Send_two_pos THEN
			uiSignalOutControl := 0;
			NewState := 95;
		END_IF

	95:
		IF uiSignalInAck = 0 THEN
			gResetPcCom := TRUE;
			NewState := 100;
		END_IF


	100:		(* Retry Grab Stem *)
		FB_RETRY_GRAB_STEM.Execute := TRUE;
		uiSignalOutControl := FB_RETRY_GRAB_STEM.OutQ;
		IF FB_RETRY_GRAB_STEM.Done THEN
			FB_RETRY_GRAB_STEM.Execute := FALSE;
			gResetPcCom := TRUE;
			NewState := 20;
		END_IF


	1000:
		Done := TRUE;
		IF NOT Execute THEN
			Fail := FALSE;
			bRetry := 0;
			NewState := 0;
		END_IF



END_CASE

bRobotFail := uiSignalIn2.07;

END_FUNCTION_BLOCK

// ---- POUs/SEQUENCEs/MoveOnStem.TcPOU
FUNCTION_BLOCK MoveOnStem
VAR_INPUT
	Execute: 		BOOL;
	State : 		INT;
	NewState : 	INT;

END_VAR
VAR_OUTPUT


END_VAR
VAR


	Done: 		BOOL;
	Fail: BOOL;
	bRetry: USINT;
	JointReached: BOOL;
	Height: UINT;
	iCnfgChange: USINT;
	bRobotFail: BOOL;
END_VAR

IF State <> NewState THEN
	State := NewState;
END_IF

CASE  State OF
	0:
		Done := FALSE;
		IF Execute  THEN
			NewState	 :=10;
		END_IF

	10:		(* Send Robot Pick Position *)
		getPickCoords := TRUE;
		IF bPosSentToPcCom AND FB_GET_PICK_COORD.Execute = FALSE THEN
			ImageRetryHeight := stDataToVision.CoordZR2G;
			bPosSentToPcCom := FALSE;
			bGetCoordDone := FALSE;
			NewState := 20;
		END_IF

	20:
		IF stDataToVision.CoordXR2G <> 0 AND stDataToVision.CoordYR2G <> 0 AND stDataToVision.CoordZR2G <> 0 THEN
			FB_CAM_TWO_CONTROL.Execute := TRUE;
			IF FB_CAM_TWO_CONTROL.Done THEN
				FB_CAM_TWO_CONTROL.Execute := FALSE;
				(* Check if the stem is found *)
				IF FB_CAM_TWO_CONTROL.StemFound = 1 THEN
					GviX := (FB_CAM_TWO_CONTROL.X + 320) / 2;
					GviY := (FB_CAM_TWO_CONTROL.Y + 320) / 2;
					GviZ := FB_CAM_TWO_CONTROL.Z;
					Height := FB_CAM_TWO_CONTROL.Z;
					GviA := 0;
					GviE := 0;
					GviR := 40;
					IF FB_CAM_TWO_CONTROL.JointFound = 1 THEN
						GviPick := FB_CAM_TWO_CONTROL.PickAngle;
						iImageZone := FB_CAM_TWO_CONTROL.Zone;
						gResetPcCom := TRUE;
						JointReached := TRUE;
						NewState := 1000;
					ELSE
						gResetPcCom := TRUE;
						NewState := 30;
					END_IF
				ELSE
					gResetPcCom := TRUE;
					NewState := 500;
				END_IF
			END_IF
		END_IF

	30:		(* Send coordinates *)
		(* Send pos to Robots *)
		(* GsendCoord			-->	Starter SendCoordinates sekvensen							-	Sender koordinater til robotterne 		*)
		(* uiSignalOutShared.06	-->	Bekræftelse på at koordinaterne er sendt til udgangene i box 10	-	Acknowledge fra SendCoordinates	*)
		GsendCoord := TRUE;
		IF uiSignalOutShared.06 THEN
			(* Send_pos	-->	Kommando der fortæller robot cut at nogle nye positioner er sendt *)
			uiSignalOutControl := Send_pos;
		END_IF
		IF uiSignalInAck = Send_pos THEN
			uiSignalOutControl := 0;
			uiCalibImgCount := uiCalibImgCount + 1;
			NewState := 35;
		END_IF

	35:
		IF uiSignalInAck = 0 THEN
			NewState := 40;
		END_IF

	40:		(* CO-MOVE up the stem *)
		FB_COMOVE_IMAGE.Execute := TRUE;
		uiSignalOutControl := FB_COMOVE_IMAGE.OutQ;
		IF FB_COMOVE_IMAGE.Done THEN
			FB_COMOVE_IMAGE.Execute := FALSE;
			IF bRobotFail THEN
				NewState := 600;
			ELSE
				NewState := 50;
			END_IF
		END_IF

	50:		(* Send Pick coordinate *)
		(* Send Pick pos to PcCom for next image *)
		getPickCoords := TRUE;
		IF bPosSentToPcCom AND FB_GET_PICK_COORD.Execute = FALSE THEN
			bPosSentToPcCom := FALSE;
			IF Height < iBunchPosZ THEN
				NewState := 20;
			ELSE
				NewState := 1000;
			END_IF
		END_IF



	500:		(* Stem cannot be found		-->		Change configuration *)
		(* Change configuration *)
		iCnfgChange := iCnfgChange + 1;
		IF uiCalibImgCount >= 50 AND uiCalibImgCount <= 200 THEN
			NewState := 505;
		ELSIF uiCalibImgCount = 250 THEN
			bBackToZero := TRUE;
		END_IF
		gResetPcCom := TRUE;
		NewState := 505;

	505:
		IF iCnfgChange <= 5 THEN
			uiCalibImgCount := INT_TO_BYTE(iCnfgChange * 50);
		ELSE
			bBackToZero := TRUE;
		END_IF
		(* Robot Pick to image pos *)
		FB_PICK_TRUNK_IMAGE.Execute := TRUE;
		uiSignalOutControl := FB_PICK_TRUNK_IMAGE.OutQ;
		IF FB_PICK_TRUNK_IMAGE.Done THEN
			FB_PICK_TRUNK_IMAGE.Execute := FALSE;
			NewState := 510;
		END_IF

	510:		(* Send Pick coordinate *)
		(* Send Pick pos to PcCom for next image *)
		getPickCoords := TRUE;
		IF bPosSentToPcCom THEN
			bPosSentToPcCom := FALSE;
			NewState := 20;
		END_IF




	600:		(* Robot cut reached either stick-out or joint *)
		(* Get Cut coord *)
		getCutCoords := TRUE;
		IF bPosSentToPcCom AND FB_GET_CUT_COORD.Execute = FALSE THEN
			bPosSentToPcCom := FALSE;
			gResetPcCom := TRUE;
			NewState := 605;
		END_IF

	605:
		IF uiSignalInAck = 0 THEN
			uiCutCoordX	:= stDataToVision.CoordXR1G / 10;
			uiCutCoordY	:= stDataToVision.CoordYR1G / 10;
			uiCutCoordZ	:= stDataToVision.CoordZR1G / 10;

			NewState := 610;
		END_IF

	610:
		GviX := uiCutCoordX;
		GviY := uiCutCoordY;
		GviZ := uiCutCoordZ;
		GviA := 0;
		GviE := 0;
		GviR := 40;

		IF uiCutCoordZ > iBunchPosZ THEN
			(* Then cut must have reached the joint*)

			(* Send pos to Robots *)
			(* GsendCoord			-->	Starter SendCoordinates sekvensen							-	Sender koordinater til robotterne 		*)
			(* uiSignalOutShared.06	-->	Bekræftelse på at koordinaterne er sendt til udgangene i box 10	-	Acknowledge fra SendCoordinates	*)
			GsendCoord := TRUE;
			IF uiSignalOutShared.06 THEN
				(* Send_pos	-->	Kommando der fortæller robot cut at nogle nye positioner er sendt *)
				uiSignalOutControl := Send_pos;
			END_IF
			IF uiSignalInAck = Send_pos THEN
				uiSignalOutControl := 0;
				uiCalibImgCount := uiCalibImgCount + 1;
				NewState := 615;
			END_IF

		ELSE
			(* It must be a too big of a stick-out *)
			FB_RELEASE_CUT.Execute := TRUE;
			IF FB_RELEASE_CUT.Done THEN
				FB_RELEASE_CUT.Execute := FALSE;
				NewState := 630;
			END_IF
		END_IF

	615:
		IF uiSignalInAck = 0 THEN
			JointReached := TRUE;
			NewState := 620;
		END_IF

	620:
		FB_COMOVE_IMAGE.Execute := TRUE;
		uiSignalOutControl := FB_COMOVE_IMAGE.OutQ;
		IF FB_COMOVE_IMAGE.Done THEN
			FB_COMOVE_IMAGE.Execute := FALSE;
			NewState := 900;
			JointReached := TRUE;
		END_IF

	630:
		FB_LOAD_CUT.Execute := TRUE;
		IF FB_LOAD_CUT.Done THEN
			FB_LOAD_CUT.Execute := FALSE;
			NewState := 10;
		END_IF





	900:
		(* Send Pick pos to PcCom for next image *)
		getPickCoords := TRUE;
		IF bPosSentToPcCom AND FB_GET_PICK_COORD.Execute = FALSE THEN
			bPosSentToPcCom := FALSE;
			NewState := 1000;
		END_IF


	1000:
		Done := TRUE;
		IF NOT Execute THEN
			Fail := FALSE;
			bRetry := 0;
			JointReached := FALSE;
			Height := 0;
			iCnfgChange := 0;
			NewState := 0;
		END_IF



END_CASE
bRobotFail := uiSignalIn2.07;

END_FUNCTION_BLOCK

// ---- POUs/SEQUENCEs/FindJoint.TcPOU
 FUNCTION_BLOCK FindJoint
VAR_INPUT
	Execute: 		BOOL;
	State : 		INT;
	NewState : 	INT;

END_VAR
VAR_OUTPUT


END_VAR
VAR


	Done: 		BOOL;
	Fail: BOOL;
	bRetry: INT;
	bRobotFail: BOOL;
	iCnfgChange: INT;
END_VAR

IF State <> NewState THEN
	State := NewState;
END_IF

CASE  State OF
	0:
		Done := FALSE;
		IF Execute  THEN
			gResetPcCom := TRUE;
			NewState	 :=10;
		END_IF

	10:		(* Send Robot Pick Position *)
		getPickCoords := TRUE;
		IF bPosSentToPcCom AND FB_GET_PICK_COORD.Execute = FALSE THEN
			ImageRetryHeight := stDataToVision.CoordZR2G;
			bPosSentToPcCom := FALSE;
			bGetCoordDone := FALSE;
			NewState := 20;
		END_IF

	20:		(* Take a picture *)
		IF stDataToVision.CoordXR2G <> 0 AND stDataToVision.CoordYR2G <> 0 AND stDataToVision.CoordZR2G <> 0 THEN
			FB_CAM_TWO_CONTROL.Execute := TRUE;
			IF FB_CAM_TWO_CONTROL.Done THEN
				IF FB_CAM_TWO_CONTROL.StemFound <> 1 THEN
					(* Change configuration *)
					(* IF cnfgCount <> 0 THEN *)
					FB_CAM_TWO_CONTROL.Execute := FALSE;
					NewState := 100;
				ELSE
					IF FB_CAM_TWO_CONTROL.JointFound <> 1 THEN
						(* MOVE ON STEM *)
						GviX := (FB_CAM_TWO_CONTROL.X + 320) / 2;
						GviY := (FB_CAM_TWO_CONTROL.Y + 320) / 2;
						GviZ := FB_CAM_TWO_CONTROL.Z;
						GviA 	:= 0;
						GviE 	:= 0;
						GviR 	:= 40;

						FB_CAM_TWO_CONTROL.Execute := FALSE;
						gResetPcCom := TRUE;
						NewState := 50;

					ELSE
						IF FB_CAM_TWO_CONTROL.PickAngle = 0 THEN
							(* MOVE ON STEM *)
							GviX := (FB_CAM_TWO_CONTROL.X + 320) / 2;
							GviY := (FB_CAM_TWO_CONTROL.Y + 320) / 2;
							GviZ := FB_CAM_TWO_CONTROL.Z;
							GviA 	:= 0;
							GviE 	:= 0;
							GviR 	:= 40;
	
							FB_CAM_TWO_CONTROL.Execute := FALSE;
							gResetPcCom := TRUE;
							NewState := 50;
						ELSE
							(* SEND CUT COORD + HEADING *)
							GviPick := FB_CAM_TWO_CONTROL.PickAngle;
							(* Get Cut coord *)
							getCutCoords := TRUE;
							IF bPosSentToPcCom AND FB_GET_CUT_COORD.Execute = FALSE THEN
								bPosSentToPcCom := FALSE;
								FB_CAM_TWO_CONTROL.Execute := FALSE;
								gResetPcCom := TRUE;
								NewState := 25;
							END_IF
						END_IF
					END_IF
				END_IF
			END_IF
		END_IF

	25:
		IF uiSignalInAck = 0 THEN
			GviX	:= stDataToVision.CoordXR1G / 10;
			GviY	:= stDataToVision.CoordYR1G / 10;
			GviZ	:= stDataToVision.CoordZR1G / 10;
			gResetPcCom := TRUE;
			NewState := 30;
		END_IF

	30:		(* Send pos *)
		(* GsendCoord			-->	Starter SendCoordinates sekvensen							-	Sender koordinater til robotterne 		*)
		(* uiSignalOutShared.06	-->	Bekræftelse på at koordinaterne er sendt til udgangene i box 10	-	Acknowledge fra SendCoordinates	*)
		GsendCoord := TRUE;
		IF uiSignalOutShared.06 THEN
			(* Send_pos	-->	Kommando der fortæller robot cut at nogle nye positioner er sendt *)
			uiSignalOutControl := Send_pos;
		END_IF
		IF uiSignalInAck = Send_pos THEN
			uiSignalOutControl := 0;
			(*uiCalibImgCount := uiCalibImgCount + 1;*)
			NewState := 35;
		END_IF

	35:
		IF uiSignalInAck = 0 THEN
			NewState := 1000;
		END_IF


	(* ------------------------------------------------------------------------------------- *)

	50:		(* Send pos *)
		(* GsendCoord			-->	Starter SendCoordinates sekvensen							-	Sender koordinater til robotterne 		*)
		(* uiSignalOutShared.06	-->	Bekræftelse på at koordinaterne er sendt til udgangene i box 10	-	Acknowledge fra SendCoordinates	*)
		GsendCoord := TRUE;
		IF uiSignalOutShared.06 THEN
			(* Send_pos	-->	Kommando der fortæller robot cut at nogle nye positioner er sendt *)
			uiSignalOutControl := Send_pos;
		END_IF
		IF uiSignalInAck = Send_pos THEN
			uiSignalOutControl := 0;
			(*uiCalibImgCount := uiCalibImgCount + 1;*)
			NewState := 55;
		END_IF

	55:
		IF uiSignalInAck = 0 THEN
			NewState := 60;
		END_IF

	60:
		FB_COMOVE_IMAGE.Execute := TRUE;
		uiSignalOutControl := FB_COMOVE_IMAGE.OutQ;
		IF FB_COMOVE_IMAGE.Done THEN
			IF bRobotFail THEN
				FB_COMOVE_IMAGE.Execute := FALSE;
				NewState := 70;
			ELSE
				FB_COMOVE_IMAGE.Execute := FALSE;
				NewState := 10;
			END_IF
		END_IF

	70:
		(* Get Cut coord *)
		getCutCoords := TRUE;
		IF bPosSentToPcCom AND FB_GET_CUT_COORD.Execute = FALSE THEN
			bPosSentToPcCom := FALSE;
			FB_CAM_TWO_CONTROL.Execute := FALSE;
			gResetPcCom := TRUE;
			NewState := 25;
		END_IF


	(* ------------------------------------------------------------------------------------- *)

	100:		(* Stem cannot be found		-->		Change configuration *)
		(* Change configuration *)
		iCnfgChange := iCnfgChange + 1;
		IF uiCalibImgCount >= 50 AND uiCalibImgCount <= 200 THEN
			gResetPcCom := TRUE;
			NewState := 105;
		ELSIF uiCalibImgCount = 250 THEN
			Fail := TRUE;
			NewState := 1000;
		END_IF

	105:
		IF iCnfgChange <= 5 THEN
			uiCalibImgCount := INT_TO_BYTE(iCnfgChange * 50);
		ELSE
			bBackToZero := TRUE;
		END_IF
		NewState := 110;

	110:
		(* Robot Pick to image pos *)
		FB_PICK_TRUNK_IMAGE.Execute := TRUE;
		uiSignalOutControl := FB_PICK_TRUNK_IMAGE.OutQ;
		IF FB_PICK_TRUNK_IMAGE.Done THEN
			FB_PICK_TRUNK_IMAGE.Execute := FALSE;
			NewState := 120;
		END_IF

	120:		(* Send Pick coordinate *)
		(* Send Pick pos to PcCom for next image *)
		getPickCoords := TRUE;
		IF bPosSentToPcCom AND FB_GET_PICK_COORD.Execute = FALSE THEN
			bPosSentToPcCom := FALSE;
			NewState := 20;
		END_IF


	(* ------------------------------------------------------------------------------------- *)

	1000:
		Done := TRUE;
		IF NOT Execute THEN
			Fail := FALSE;
			bRetry := 0;
			iCnfgChange := 0;
			NewState := 0;
		END_IF



END_CASE

bRobotFail := uiSignalIn2.07;

END_FUNCTION_BLOCK

// ---- POUs/SEQUENCEs/GrabJoint.TcPOU
FUNCTION_BLOCK GrabJoint
VAR_INPUT
	Execute: 		BOOL;
	State : 		INT;
	NewState : 	INT;

END_VAR
VAR_OUTPUT


END_VAR
VAR

	Done: 		BOOL;
	Fail: BOOL;
	bRetry: USINT;
	bRobotFail: BOOL;
END_VAR

IF State <> NewState THEN
	State := NewState;
END_IF

CASE  State OF
	0:
		Done := FALSE;
		IF Execute  THEN
			IF uimodeNo = 2 THEN
				NewState 	:= 20;
			ELSE
				NewState	 :=10;
			END_IF
		END_IF

	10:		(* Robot Pick grab *)
		FB_PICK_GRAB.Execute := TRUE;
		uiSignalOutControl := FB_PICK_GRAB.OutQ;
		IF FB_PICK_GRAB.Done THEN
			FB_PICK_GRAB.Execute := FALSE;
			IF NOT bRobotFail THEN
				bRetry := 0;
				NewState := 20;
			ELSE
				IF bRetry = 0 THEN
					(* Take a new picture *)

					bRetry := 1;
					NewState := 500;
				ELSE
					Fail := TRUE;
				END_IF
			END_IF
		END_IF

	20:		(* Cut *)
		FB_RELEASE_CUT.Execute := TRUE;
		IF FB_RELEASE_CUT.Done THEN
			FB_RELEASE_CUT.Execute := FALSE;
			NewState := 25;
		END_IF

	25:		(* Load Cut *)
		FB_LOAD_CUT.Execute := TRUE;
		IF FB_LOAD_CUT.Done THEN
			FB_LOAD_CUT.Execute := FALSE;
			IF uimodeNo <= 1 THEN
				NewState := 30;
			ELSE
				NewState := 1000;
			END_IF
		END_IF

	30:		(* Move from pick *)
		FB_PICK_MOVE_FROM_PICK.Execute := TRUE;
		uiSignalOutControl := FB_PICK_MOVE_FROM_PICK.OutQ;
		IF FB_PICK_MOVE_FROM_PICK.Done THEN
			FB_PICK_MOVE_FROM_PICK.Execute := FALSE;
			NewState := 1000;
		END_IF

	500:
		FB_RETRY_GRAB_STEM.Execute := TRUE;
		IF FB_RETRY_GRAB_STEM.Done THEN
			FB_RETRY_GRAB_STEM.Execute := FALSE;
			NewState := 1000;
		END_IF


	1000:
		Done := TRUE;
		IF NOT Execute THEN
			IF Fail THEN
				bRetry := 0;
				Fail := FALSE;
			END_IF
			NewState := 0;
		END_IF



END_CASE

bRobotFail := uiSignalIn2.07;

END_FUNCTION_BLOCK

// ---- POUs/SEQUENCEs/DeleafPlace.TcPOU
FUNCTION_BLOCK DeleafPlace
VAR_INPUT
	Execute: 		BOOL;
	State : 		INT;
	NewState : 	INT;

END_VAR
VAR_OUTPUT


END_VAR
VAR

	Done: 		BOOL;
	Fail: BOOL;
	bRetry: USINT;
	iMoved: USINT;
	uiDeleaf: USINT;
END_VAR

IF State <> NewState THEN
	State := NewState;
END_IF

CASE  State OF
	0:
		Done := FALSE;
		IF Execute  THEN
			IF uimodeNo = 1 THEN
				NewState := 40;
			ELSE
				NewState	 :=10;
			END_IF
		END_IF

	10:		(* Image of LEAFS *)
		uiCalibImgCount := INT_TO_BYTE(iMoved * 50);
		FB_PICK_DELEAF_PROGRAM.Execute := TRUE;
		uiSignalOutControl := FB_PICK_DELEAF_PROGRAM.OutQ;
		IF FB_PICK_DELEAF_PROGRAM.Done THEN
			iMoved := iMoved + 1;
			FB_PICK_DELEAF_PROGRAM.Execute := FALSE;
			NewState := 20;
		END_IF

	20:		(* Send Pick coordinate *)
		getPickCoords := TRUE;
		IF bPosSentToPcCom AND FB_GET_PICK_COORD.Execute = FALSE THEN
			bPosSentToPcCom := FALSE;
			NewState := 30;
		END_IF

	30:
		IF stDataToVision.CoordXR2G <> 0 AND stDataToVision.CoordYR2G <> 0 AND stDataToVision.CoordZR2G <> 0 THEN
			FB_CAM_TWO_CONTROL.Execute := TRUE;
			IF FB_CAM_TWO_CONTROL.Done THEN
				IF FB_CAM_TWO_CONTROL.StemFound = 1 THEN
					IF FB_CAM_TWO_CONTROL.PickAngle <> 0 AND FB_CAM_TWO_CONTROL.JointFound = 1 THEN
						GviX 		:= FB_CAM_TWO_CONTROL.X;
						GviY 		:= FB_CAM_TWO_CONTROL.Y;
						GviZ 		:= FB_CAM_TWO_CONTROL.Z;
						GviA 		:= 0;
						GviE 		:= 0;
						GviR 		:= 40;
						GviPick 		:= FB_CAM_TWO_CONTROL.PickAngle;
						iImageZone 	:= FB_CAM_TWO_CONTROL.Zone;
						gJointFound 	:= FB_CAM_TWO_CONTROL.JointFound;

						FB_CAM_TWO_CONTROL.Execute := FALSE;
						gResetPcCom := TRUE;
						NewState := 40;

					ELSE
						FB_CAM_TWO_CONTROL.Execute := FALSE;
						gResetPcCom := TRUE;
						NewState := 10;

					END_IF
				ELSE
					FB_CAM_TWO_CONTROL.Execute := FALSE;
					gResetPcCom := TRUE;
					NewState := 10;
				END_IF
			END_IF
		END_IF

	40:		(* Send pos *)
		IF uiModeNo = 0 AND uiDeleaf  = 0 THEN
			FB_PLACE.Execute := TRUE;
			IF FB_PLACE.Done THEN
				GviX2 := FB_PLACE.X;
				GviY2 := FB_PLACE.Y;
				GviZ2 := FB_PLACE.Z;
				(* GsendCoord			-->	Starter SendCoordinates sekvensen							-	Sender koordinater til robotterne 		*)
				(* uiSignalOutShared.06	-->	Bekræftelse på at koordinaterne er sendt til udgangene i box 10	-	Acknowledge fra SendCoordinates	*)
				GsendCoord := TRUE;
				IF uiSignalOutShared.06 THEN
					(* Send_pos	-->	Kommando der fortæller robot cut at nogle nye positioner er sendt *)
					uiSignalOutControl := Send_two_pos;
				END_IF
				IF uiSignalInAck = Send_two_pos THEN
					uiSignalOutControl := 0;
					uiCalibImgCount := uiCalibImgCount + 1;
					FB_PLACE.Execute := FALSE;
					NewState := 45;
				END_IF
			END_IF
		ELSIF uiModeNo = 1 AND uiDeleaf  = 0 THEN
			FB_PLACE.Execute := TRUE;
			IF FB_PLACE.Done THEN
				GviX := FB_PLACE.X;
				GviY := FB_PLACE.Y;
				GviZ := FB_PLACE.Z;
				(* GsendCoord			-->	Starter SendCoordinates sekvensen							-	Sender koordinater til robotterne 		*)
				(* uiSignalOutShared.06	-->	Bekræftelse på at koordinaterne er sendt til udgangene i box 10	-	Acknowledge fra SendCoordinates	*)
				GsendCoord := TRUE;
				IF uiSignalOutShared.06 THEN
					(* Send_pos	-->	Kommando der fortæller robot cut at nogle nye positioner er sendt *)
					uiSignalOutControl := Send_pos;
				END_IF
				IF uiSignalInAck = Send_pos THEN
					uiSignalOutControl := 0;
					uiCalibImgCount := uiCalibImgCount + 1;
					FB_PLACE.Execute := FALSE;
					NewState := 45;
				END_IF
			END_IF
		ELSIF uiModeNo = 2 OR uiDeleaf  > 0 THEN
			(* GsendCoord			-->	Starter SendCoordinates sekvensen							-	Sender koordinater til robotterne 		*)
			(* uiSignalOutShared.06	-->	Bekræftelse på at koordinaterne er sendt til udgangene i box 10	-	Acknowledge fra SendCoordinates	*)
			GsendCoord := TRUE;
			IF uiSignalOutShared.06 THEN
				(* Send_pos	-->	Kommando der fortæller robot cut at nogle nye positioner er sendt *)
				uiSignalOutControl := Send_pos;
			END_IF
			IF uiSignalInAck = Send_pos THEN
				uiSignalOutControl := 0;
				uiCalibImgCount := uiCalibImgCount + 1;
				FB_PLACE.Execute := FALSE;
				NewState := 45;
			END_IF
		END_IF



	45:
		IF uiSignalInAck = 0 THEN
			NewState := 50;
		END_IF

	50:
		IF uimodeNo = 0 AND uiDeleaf  = 0 THEN
			FB_PLACE_DELEAF.Execute := TRUE;
			uiSignalOutControl := FB_PLACE_DELEAF.OutQ;
			IF FB_PLACE_DELEAF.Done THEN
				FB_PLACE_DELEAF.Execute := FALSE;
				NewState := 80;
			END_IF
		ELSIF uimodeNo = 1 AND uiDeleaf  = 0 THEN
			FB_PICK_PLACE.Execute := TRUE;
			uiSignalOutControl := FB_PICK_PLACE.OutQ;
			IF FB_PICK_PLACE.Done THEN
				FB_PICK_PLACE.Execute := FALSE;
				NewState := 1000;
			END_IF
		ELSE
			FB_PICK_DELEAF_PROGRAM.Execute := TRUE;
			uiSignalOutControl := FB_PICK_DELEAF_PROGRAM.OutQ;
			IF FB_PICK_DELEAF_PROGRAM.Done THEN
				FB_PICK_DELEAF_PROGRAM.Execute := FALSE;
				NewState := 80;
			END_IF
		END_IF


	80:		(* Load Cut *)
		FB_LOAD_CUT.Execute := TRUE;
		IF FB_LOAD_CUT.Done THEN
			FB_LOAD_CUT.Execute := FALSE;
			NewState := 85;
		END_IF

	85:
		IF uiDeleaf < 0 THEN
			uiDeleaf := uiDeleaf + 1;
			NewState := 10;
		ELSE
			uiDeleaf := 0;
			NewState := 1000;
		END_IF


	1000:
		Done := TRUE;
		IF NOT Execute THEN
			bRetry := 0;
			Fail := FALSE;
			NewState := 0;
		END_IF



END_CASE

END_FUNCTION_BLOCK

// ---- POUs/FUNCTIONs/ValveControl_1.TcPOU
FUNCTION_BLOCK ValveControl_1
VAR_INPUT
	ControlType: 	USINT;		(*	1: Controlling valves from Robot		2: Controlling valves from Robot and  PLC		3: Close only using PLC		4: Open only using PLC		*)
	Ack: 			BOOL;
	Execute: 		BOOL;
	ExecuteHmi:		BOOL;

END_VAR
VAR_OUTPUT
	OutQ: 		BOOL;
	OutQ2: 		BOOL;
	OutQ3: 		BOOL;
END_VAR
VAR
	WaitValve:	TON;

	State: 		INT;
	NewState: 	INT;

	Done: 		BOOL;
	bValveTime: 	BOOL;
END_VAR

IF State <> NewState THEN
	State := NewState;
END_IF

CASE  State OF
	0:
		Done := FALSE;
		IF Execute THEN
			IF ControlType = 1 THEN
				NewState	 :=10;
			ELSIF ControlType = 2 OR ControlType = 5 THEN
				NewState := 100;
			ELSIF ControlType = 3 OR ControlType = 4 THEN
				NewState := 200;
			ELSE
				NewState := 0;
			END_IF
		ELSIF ExecuteHmi THEN
			//ExecuteHmi := FALSE;
			IF ControlType = 1 THEN
				NewState	 :=10;
			ELSIF ControlType = 2 OR ControlType = 5 THEN
				NewState := 100;
			ELSIF ControlType = 3 OR ControlType = 4 THEN
				NewState := 200;
			ELSE
				NewState := 0;
			END_IF
		END_IF

	10:
		OutQ := TRUE;
		IF Ack THEN
			OutQ := FALSE;
			NewState := 1000;
		END_IF

	100:
		OutQ2 := TRUE;
		bValveTime := TRUE;
		IF waitValve.Q THEN
			bValveTime := FALSE;
			NewState 	:=110;
		END_IF

	110:

		OutQ := TRUE;
		IF Ack THEN
			OutQ := FALSE;
			NewState := 120;
		END_IF

	120:
		OutQ2 := FALSE;
		IF ControlType = 5 THEN
			NewState := 130;
		ELSE
			NewState := 140;
		END_IF
		
	130:
		OutQ3 := TRUE;
		bValveTime := TRUE;
		IF waitValve.Q THEN
			bValveTime := FALSE;
			NewState 	:=140;
		END_IF
		
	140:
		//OutQ3 := FALSE;
		bValveTime := TRUE;
		IF waitValve.Q THEN
			OutQ3 := FALSE;
			bValveTime := FALSE;
			NewState 	:= 1000;
		END_IF

	200:
		IF ControlType = 3 THEN
			OutQ := TRUE;
			bValveTime := TRUE;
			IF waitValve.Q THEN
				bValveTime := FALSE;
				NewState 	:=1000;
			END_IF
		ELSE
			OutQ := TRUE;
			bValveTime := TRUE;
			IF waitValve.Q THEN
				bValveTime := FALSE;
				NewState 	:=1000;
			END_IF
		END_IF

	1000:
		Done := TRUE;
		IF NOT Execute THEN
			NewState := 0;
		END_IF



END_CASE

(* Timer *)
WaitValve		(IN:=  bValveTime		, PT:=T#1500MS, Q=>, ET=>); 		(*Timer*)		(* For waiting for Valves 			*)

END_FUNCTION_BLOCK
